{attribute 'linkalways'} 
{attribute 'no_explicit_call' := 'This FB is a CLASS and must be accessed using methods or properties'}
{attribute 'enable_dynamic_creation'}
FUNCTION_BLOCK _ETcVnFeatureScalingType EXTENDS EnumDatatypeBase
VAR
	localData : ETcVnFeatureScalingType;
	activeData : REFERENCE TO ETcVnFeatureScalingType;
	enumBaseDatatype : _DINT(localData);
END_VAR

METHOD PRIVATE AddLocalEnumeration
VAR_INPUT
	Enumeration : T_MAXSTRING;
	Value : ETcVnFeatureScalingType;
END_VAR
AddEnumeration(Enumeration, Value);
END_METHOD

PROPERTY PUBLIC Address : PVOID
GET
Address := ADR(activeData);
END_GET
END_PROPERTY

METHOD PUBLIC ClearReference
VAR_INPUT
END_VAR
activeData REF= localData;
SetBaseDatatypeReference();
END_METHOD

METHOD PUBLIC Clone : I_Datatype
VAR
    pClone : POINTER TO _ETcVnFeatureScalingType;
END_VAR
pClone := __NEW(_ETcVnFeatureScalingType(InitialValue := Value));
Clone := pClone^;
END_METHOD

METHOD FB_init : BOOL
VAR_INPUT
	bInitRetains : BOOL; // if TRUE, the retain variables are initialized (warm start / cold start)
	bInCopyCode : BOOL;  // if TRUE, the instance afterwards gets moved into the copy code (online change)
	InitialValue : ETcVnFeatureScalingType;
END_VAR
localData := InitialValue;
AddBaseDatatype(enumBaseDatatype);
ClearReference();

AddLocalEnumeration('TCVN_FST1_MAXABS', ETcVnFeatureScalingType.TCVN_FST1_MAXABS);
AddLocalEnumeration('TCVN_FST1_MINMAX', ETcVnFeatureScalingType.TCVN_FST1_MINMAX);
AddLocalEnumeration('TCVN_FST1_STANDARDIZATION', ETcVnFeatureScalingType.TCVN_FST1_STANDARDIZATION);
END_METHOD

PROPERTY PUBLIC Identifier : T_MAXSTRING
GET
Identifier := 'ETcVnFeatureScalingType';
END_GET
END_PROPERTY

METHOD IsEnumeratorValueEqual : BOOL
VAR_INPUT
	Enumerator : I_KeyValueForwardEnumerator;
END_VAR
VAR
	storedValue : ETcVnFeatureScalingType;
END_VAR
IF NOT Enumerator.TryGet(storedValue) THEN
	RETURN;
END_IF

IsEnumeratorValueEqual := storedValue = activeData;
END_METHOD

METHOD PUBLIC MakeReferenceTo
VAR_INPUT
	ReferenceTarget : REFERENCE TO ETcVnFeatureScalingType;
END_VAR
activeData REF= ReferenceTarget;
SetBaseDatatypeReference();
END_METHOD

METHOD PROTECTED SetBaseDatatypeReference
VAR_INPUT
END_VAR
enumBaseDatatype.MakeReferenceTo(activeData);
END_METHOD

PROPERTY PUBLIC Size : UDINT
GET
Size := SIZEOF(activeData);
END_GET
END_PROPERTY

METHOD TryMakeReferenceTo : BOOL
VAR_INPUT
	Target : I_Datatype;
END_VAR
VAR
	pTargetData : POINTER TO ETcVnFeatureScalingType;
END_VAR
IF NOT IsEquivalentTo(Target) THEN
	RETURN;
END_IF

pTargetData := Target.Address;
activeData REF= pTargetData^;
SetBaseDatatypeReference();
TryMakeReferenceTo := TRUE;
END_METHOD

PROPERTY PUBLIC Value : ETcVnFeatureScalingType
GET
Value := activeData;
END_GET
SET
activeData := Value;
END_SET
END_PROPERTY

END_FUNCTION_BLOCK

(* stored: Version 1.1.0.1, ProductVersion 3.1.4024.13
   POU _ETcVnFeatureScalingType: Id {70df1f6e-2a36-017f-1bc4-2c20cd0149af}, SpecialFunc None
   Folder Core: Id {a10def05-4041-018d-342a-225c1b881a55}
   Folder Protected: Id {f2cffdf7-e3f2-000d-3b0e-b4dbf30d1858}
   Folder Customize: Id {231a0ef6-b020-08fc-0e19-00a09e58e882}
   Folder Constructor: Id {7c7f56e0-3589-0463-1832-a3ba2b10ea53}
   Folder Private: Id {a008303e-281a-0f78-1b46-c83332f2a1de}
   Folder Protected: Id {c193fc5d-06ff-0680-2ef4-e79d03c4ca6b}
   Method AddLocalEnumeration: Id {19e1ad55-76bd-0e39-2cfa-65febeb0e046}
   Property Address: Id {6787338e-6a44-01fd-17ba-53fc8756048a}
   Get Get: Id {391e6734-a1e5-0cb0-214d-5e09e14913ba}
   Method ClearReference: Id {732fba84-9a2d-0876-3369-d01a1457d9f0}
   Method Clone: Id {da488b4d-ee97-067a-2f5c-88c425dbb580}
   Method FB_init: Id {1176f4c8-73a8-06ed-042b-8c10a9cdf229}
   Property Identifier: Id {1c272d41-6da9-0be9-19f1-0c77f1cc7cb4}
   Get Get: Id {34932923-30e8-045b-151f-be7bbfa5c558}
   Method IsEnumeratorValueEqual: Id {a872ee1c-cecf-0500-2607-367a434616ab}
   Method MakeReferenceTo: Id {ec761a61-10c0-0342-11bd-fdae5f816e60}
   Method SetBaseDatatypeReference: Id {377ed493-77ca-04c5-07e9-b04a065a6d27}
   Property Size: Id {cce00d16-ce25-05ac-08d2-0bf4c9ab0256}
   Get Get: Id {6f8ad036-ccf0-0e96-3e2e-e76eb2603536}
   Method TryMakeReferenceTo: Id {7611decf-f17c-0cb1-23d6-766ee793c6a5}
   Property Value: Id {b076bf71-76d1-012a-2ec5-d9e3c2e1191f}
   Get Get: Id {2dae3009-0426-0bf3-0aff-7d97d938fcfc}
   Set Set: Id {1ca49788-4eb6-051d-1e4d-65623605610e} *)
